Omron CX-Programmer project NewProject (CX-Programmer 9.73)

# PLC NewPLC1: CP1E E30

## Global symbols (name address type ; comment)
0.01 BOOL  ; pb start
0.02 BOOL  ; reset
100.01 BOOL  ; motor
C001 BOOL  ; counter

## Program NewProgram1 (cyclic task 0)

### Section Section1

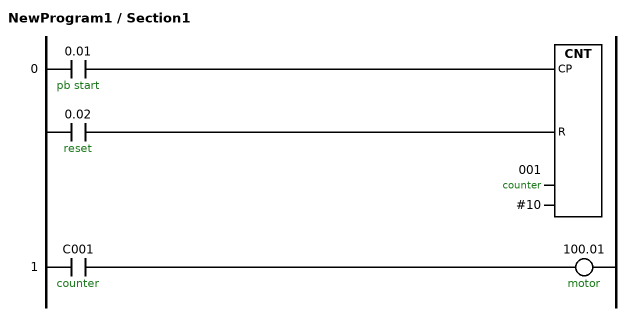
; rung 0
LD 0.01  ; pb start
LD 0.02  ; reset
CNT 001 #10  ; counter
; rung 1
LD C001  ; counter
OUT 100.01  ; motor

### Section END
; rung 0
END(001)